// TIA Portal V17 export
// export: Created 2025-03-05T08:01:12.2464352Z, ExportSetting WithDefaults, DisplayName Totally Integrated Automation Portal, DisplayVersion V17 Update 8, DisplayName TIA Portal Openness, DisplayVersion V17 Update 8, DisplayName TIA Portal Version Control Interface, DisplayVersion V17, DisplayName SINAMICS Startdrive Advanced, DisplayVersion V17 SP2, DisplayName SINAMICS Startdrive G110M, G120, G120C, G120D, G120P, G115D, DisplayVersion V17 SP2, DisplayName SINAMICS Startdrive G130, G150, S120, S150, SINAMICS MV, S210, DisplayVersion V17 SP2, DisplayName STEP 7 Professional, DisplayVersion V17 Update 8, DisplayName SINUMERIK ONE STEP 7 Toolbox, DisplayVersion V17 Update 12, DisplayName SINUMERIK 840D sl STEP 7 Toolbox, DisplayVersion V17 Update 12, DisplayName STEP 7 Safety, DisplayVersion V17 Update 6, DisplayName WinCC Advanced, DisplayVersion V17 Update 8
FUNCTION "FC2203_PROFINET_INSPEKTOR" : Void   // FC2203, LAD
{ S7_Optimized_Access := 'TRUE' }
VERSION : 0.1
// stored: AutoNumber false, IsIECCheckEnabled false, SetENOAutomatically false, UDAEnableTagReadback false
   VAR CONSTANT
      FC_NUMBER : Int := 2203;
   END_VAR
   VAR_TEMP   // added for the SCL form of the ladder/FBD networks
      _w1 : Bool;
      _w2 : Bool;
   END_VAR
BEGIN

REGION Network 1: PROFINET INSPEKTOR PROFINET FAULT INPUT
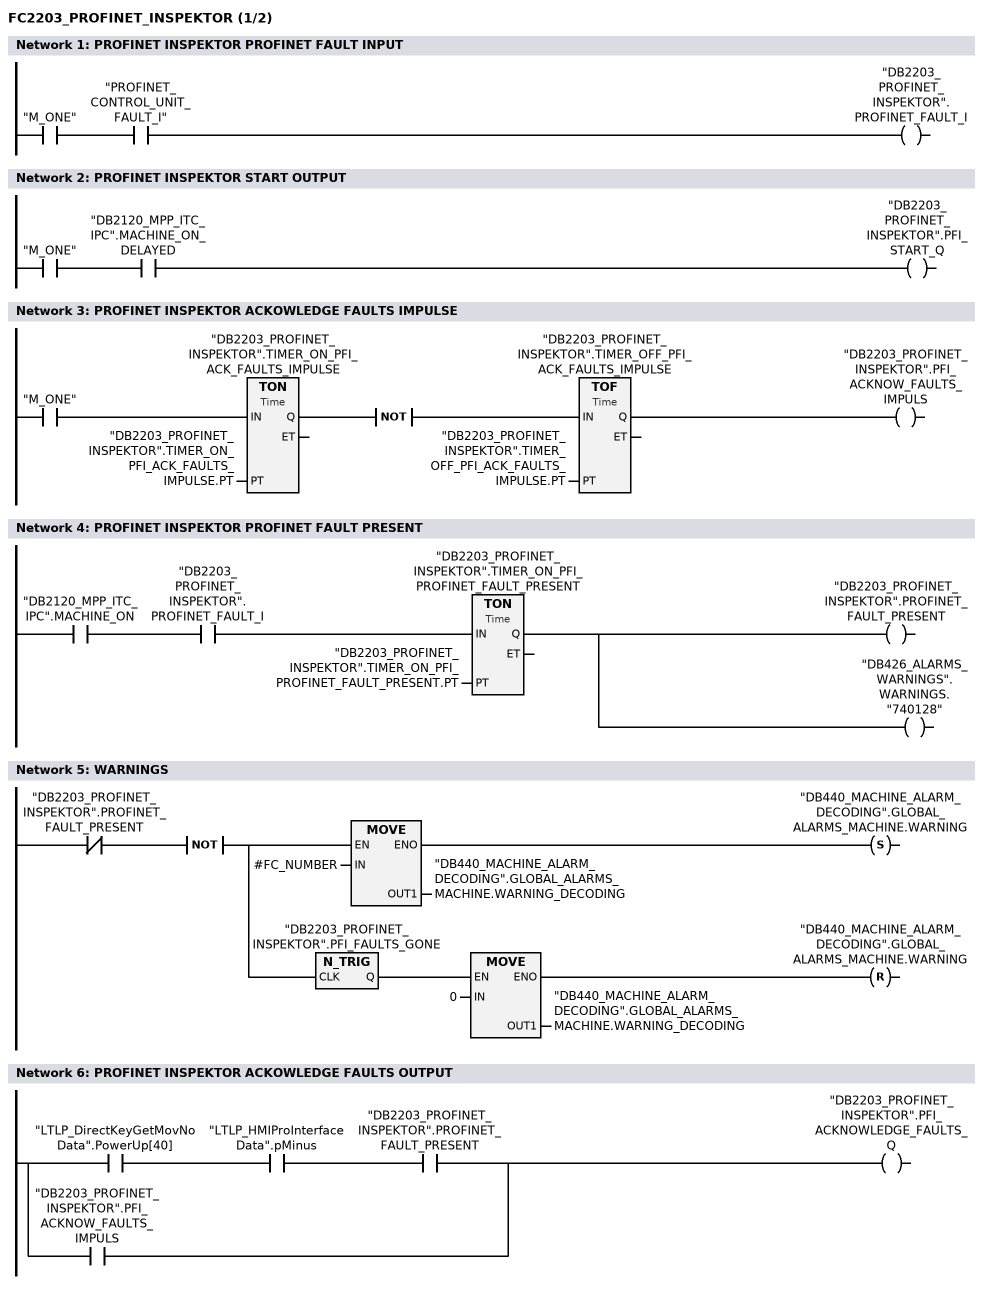
   RUNG wire#powerrail
      Contact( "M_ONE" )
      Contact( "PROFINET_CONTROL_UNIT_FAULT_I" )
      Coil( "DB2203_PROFINET_INSPEKTOR".PROFINET_FAULT_I )
   END_RUNG
   // the same network as SCL:
   "DB2203_PROFINET_INSPEKTOR".PROFINET_FAULT_I := "M_ONE" AND "PROFINET_CONTROL_UNIT_FAULT_I";
END_REGION

REGION Network 2: PROFINET INSPEKTOR START OUTPUT
   RUNG wire#powerrail
      Contact( "M_ONE" )
      Contact( "DB2120_MPP_ITC_IPC".MACHINE_ON_DELAYED )
      Coil( "DB2203_PROFINET_INSPEKTOR".PFI_START_Q )
   END_RUNG
   // the same network as SCL:
   "DB2203_PROFINET_INSPEKTOR".PFI_START_Q := "M_ONE" AND "DB2120_MPP_ITC_IPC".MACHINE_ON_DELAYED;
END_REGION

REGION Network 3: PROFINET INSPEKTOR ACKOWLEDGE FAULTS IMPULSE
   RUNG wire#powerrail
      Contact( "M_ONE" )
      { S7_Templates := "time_type := Time" } "DB2203_PROFINET_INSPEKTOR".TIMER_ON_PFI_ACK_FAULTS_IMPULSE.TON(pt := "DB2203_PROFINET_INSPEKTOR".TIMER_ON_PFI_ACK_FAULTS_IMPULSE.PT, et =>)
      Not()
      { S7_Templates := "time_type := Time" } "DB2203_PROFINET_INSPEKTOR".TIMER_OFF_PFI_ACK_FAULTS_IMPULSE.TOF(pt := "DB2203_PROFINET_INSPEKTOR".TIMER_OFF_PFI_ACK_FAULTS_IMPULSE.PT, et =>)
      Coil( "DB2203_PROFINET_INSPEKTOR".PFI_ACKNOW_FAULTS_IMPULS )
   END_RUNG
   // the same network as SCL:
   "DB2203_PROFINET_INSPEKTOR".TIMER_ON_PFI_ACK_FAULTS_IMPULSE.TON(IN := "M_ONE",
                           PT := "DB2203_PROFINET_INSPEKTOR".TIMER_ON_PFI_ACK_FAULTS_IMPULSE.PT);
   "DB2203_PROFINET_INSPEKTOR".TIMER_OFF_PFI_ACK_FAULTS_IMPULSE.TOF(IN := NOT "DB2203_PROFINET_INSPEKTOR".TIMER_ON_PFI_ACK_FAULTS_IMPULSE.Q,
                           PT := "DB2203_PROFINET_INSPEKTOR".TIMER_OFF_PFI_ACK_FAULTS_IMPULSE.PT);
   "DB2203_PROFINET_INSPEKTOR".PFI_ACKNOW_FAULTS_IMPULS := "DB2203_PROFINET_INSPEKTOR".TIMER_OFF_PFI_ACK_FAULTS_IMPULSE.Q;
END_REGION

REGION Network 4: PROFINET INSPEKTOR PROFINET FAULT PRESENT
   RUNG wire#powerrail
      Contact( "DB2120_MPP_ITC_IPC".MACHINE_ON )
      Contact( "DB2203_PROFINET_INSPEKTOR".PROFINET_FAULT_I )
      { S7_Templates := "time_type := Time" } "DB2203_PROFINET_INSPEKTOR".TIMER_ON_PFI_PROFINET_FAULT_PRESENT.TON(pt := "DB2203_PROFINET_INSPEKTOR".TIMER_ON_PFI_PROFINET_FAULT_PRESENT.PT, et =>)
      wire#w1
      Coil( "DB2203_PROFINET_INSPEKTOR".PROFINET_FAULT_PRESENT )
   END_RUNG
   RUNG wire#w1
      Coil( "DB426_ALARMS_WARNINGS".WARNINGS."740128" )
   END_RUNG
   // the same network as SCL:
   "DB2203_PROFINET_INSPEKTOR".TIMER_ON_PFI_PROFINET_FAULT_PRESENT.TON(IN := "DB2120_MPP_ITC_IPC".MACHINE_ON AND "DB2203_PROFINET_INSPEKTOR".PROFINET_FAULT_I,
                           PT := "DB2203_PROFINET_INSPEKTOR".TIMER_ON_PFI_PROFINET_FAULT_PRESENT.PT);
   "DB2203_PROFINET_INSPEKTOR".PROFINET_FAULT_PRESENT := "DB2203_PROFINET_INSPEKTOR".TIMER_ON_PFI_PROFINET_FAULT_PRESENT.Q;
   "DB426_ALARMS_WARNINGS".WARNINGS."740128" := "DB2203_PROFINET_INSPEKTOR".TIMER_ON_PFI_PROFINET_FAULT_PRESENT.Q;
END_REGION

REGION Network 5: WARNINGS
   RUNG wire#powerrail
      I_Contact( "DB2203_PROFINET_INSPEKTOR".PROFINET_FAULT_PRESENT )
      Not()
      wire#w1
      Move(in := #FC_NUMBER, out1 => "DB440_MACHINE_ALARM_DECODING".GLOBAL_ALARMS_MACHINE.WARNING_DECODING)
      S_Coil( "DB440_MACHINE_ALARM_DECODING".GLOBAL_ALARMS_MACHINE.WARNING )
   END_RUNG
   RUNG wire#w1
      N_Trig( "DB2203_PROFINET_INSPEKTOR".PFI_FAULTS_GONE )
      Move(in := 0, out1 => "DB440_MACHINE_ALARM_DECODING".GLOBAL_ALARMS_MACHINE.WARNING_DECODING)
      R_Coil( "DB440_MACHINE_ALARM_DECODING".GLOBAL_ALARMS_MACHINE.WARNING )
   END_RUNG
   // the same network as SCL:
   #_w1 := NOT (NOT "DB2203_PROFINET_INSPEKTOR".PROFINET_FAULT_PRESENT);
   IF #_w1 THEN
       "DB440_MACHINE_ALARM_DECODING".GLOBAL_ALARMS_MACHINE.WARNING_DECODING := #FC_NUMBER;
       "DB440_MACHINE_ALARM_DECODING".GLOBAL_ALARMS_MACHINE.WARNING := TRUE;
   END_IF;
   #_w2 := NOT #_w1 AND "DB2203_PROFINET_INSPEKTOR".PFI_FAULTS_GONE;   // falling edge
   "DB2203_PROFINET_INSPEKTOR".PFI_FAULTS_GONE := #_w1;
   IF #_w2 THEN
       "DB440_MACHINE_ALARM_DECODING".GLOBAL_ALARMS_MACHINE.WARNING_DECODING := 0;
       "DB440_MACHINE_ALARM_DECODING".GLOBAL_ALARMS_MACHINE.WARNING := FALSE;
   END_IF;
END_REGION

REGION Network 6: PROFINET INSPEKTOR ACKOWLEDGE FAULTS OUTPUT
   RUNG wire#powerrail
      Contact( "LTLP_DirectKeyGetMovNoData".PowerUp[40] )
      Contact( "LTLP_HMIProInterfaceData".pMinus )
      Contact( "DB2203_PROFINET_INSPEKTOR".PROFINET_FAULT_PRESENT )
      wire#w1
      Coil( "DB2203_PROFINET_INSPEKTOR".PFI_ACKNOWLEDGE_FAULTS_Q )
   END_RUNG
   RUNG wire#powerrail
      Contact( "DB2203_PROFINET_INSPEKTOR".PFI_ACKNOW_FAULTS_IMPULS )
   END_RUNG wire#w1
   // the same network as SCL:
   "DB2203_PROFINET_INSPEKTOR".PFI_ACKNOWLEDGE_FAULTS_Q := ("LTLP_DirectKeyGetMovNoData".PowerUp[40] AND "LTLP_HMIProInterfaceData".pMinus AND "DB2203_PROFINET_INSPEKTOR".PROFINET_FAULT_PRESENT) OR "DB2203_PROFINET_INSPEKTOR".PFI_ACKNOW_FAULTS_IMPULS;
END_REGION

REGION Network 7: PROFINET INSPEKTOR LOGGED DATA OUTPUT
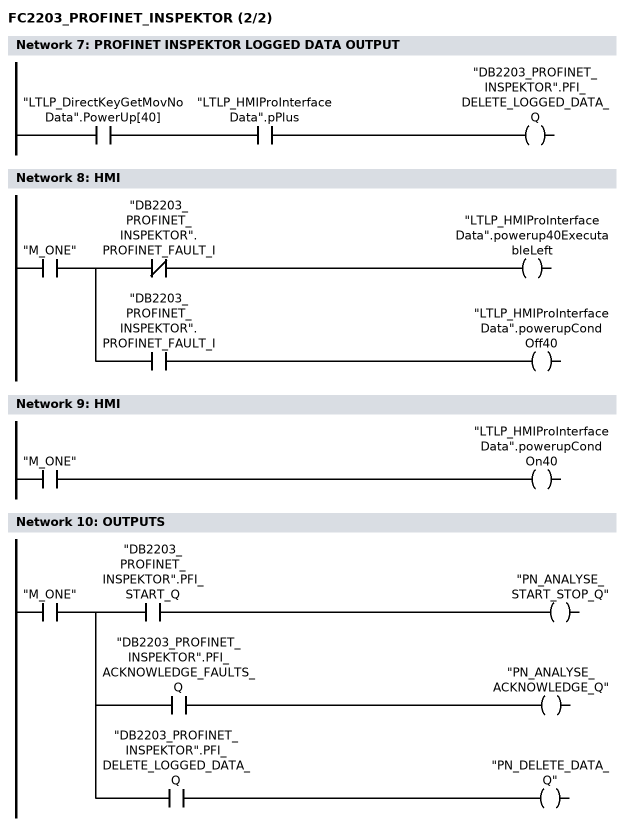
   RUNG wire#powerrail
      Contact( "LTLP_DirectKeyGetMovNoData".PowerUp[40] )
      Contact( "LTLP_HMIProInterfaceData".pPlus )
      Coil( "DB2203_PROFINET_INSPEKTOR".PFI_DELETE_LOGGED_DATA_Q )
   END_RUNG
   // the same network as SCL:
   "DB2203_PROFINET_INSPEKTOR".PFI_DELETE_LOGGED_DATA_Q := "LTLP_DirectKeyGetMovNoData".PowerUp[40] AND "LTLP_HMIProInterfaceData".pPlus;
END_REGION

REGION Network 8: HMI
   RUNG wire#powerrail
      Contact( "M_ONE" )
      wire#w1
      I_Contact( "DB2203_PROFINET_INSPEKTOR".PROFINET_FAULT_I )
      Coil( "LTLP_HMIProInterfaceData".powerup40ExecutableLeft )
   END_RUNG
   RUNG wire#w1
      Contact( "DB2203_PROFINET_INSPEKTOR".PROFINET_FAULT_I )
      Coil( "LTLP_HMIProInterfaceData".powerupCondOff40 )
   END_RUNG
   // the same network as SCL:
   "LTLP_HMIProInterfaceData".powerup40ExecutableLeft := "M_ONE" AND NOT "DB2203_PROFINET_INSPEKTOR".PROFINET_FAULT_I;
   "LTLP_HMIProInterfaceData".powerupCondOff40 := "M_ONE" AND "DB2203_PROFINET_INSPEKTOR".PROFINET_FAULT_I;
END_REGION

REGION Network 9: HMI
   RUNG wire#powerrail
      Contact( "M_ONE" )
      Coil( "LTLP_HMIProInterfaceData".powerupCondOn40 )
   END_RUNG
   // the same network as SCL:
   "LTLP_HMIProInterfaceData".powerupCondOn40 := "M_ONE";
END_REGION

REGION Network 10: OUTPUTS
   RUNG wire#powerrail
      Contact( "M_ONE" )
      wire#w1
      Contact( "DB2203_PROFINET_INSPEKTOR".PFI_START_Q )
      Coil( "PN_ANALYSE_START_STOP_Q" )
   END_RUNG
   RUNG wire#w1
      Contact( "DB2203_PROFINET_INSPEKTOR".PFI_ACKNOWLEDGE_FAULTS_Q )
      Coil( "PN_ANALYSE_ACKNOWLEDGE_Q" )
   END_RUNG
   RUNG wire#w1
      Contact( "DB2203_PROFINET_INSPEKTOR".PFI_DELETE_LOGGED_DATA_Q )
      Coil( "PN_DELETE_DATA_Q" )
   END_RUNG
   // the same network as SCL:
   "PN_ANALYSE_START_STOP_Q" := "M_ONE" AND "DB2203_PROFINET_INSPEKTOR".PFI_START_Q;
   "PN_ANALYSE_ACKNOWLEDGE_Q" := "M_ONE" AND "DB2203_PROFINET_INSPEKTOR".PFI_ACKNOWLEDGE_FAULTS_Q;
   "PN_DELETE_DATA_Q" := "M_ONE" AND "DB2203_PROFINET_INSPEKTOR".PFI_DELETE_LOGGED_DATA_Q;
END_REGION
END_FUNCTION
